// TIA Portal V18 export
FUNCTION "AHURegsAndTargetStatesInEconomyOpMode" : Void   // FC60031, LAD
{ S7_Optimized_Access := 'TRUE' }
VERSION : 0.1
// Operation Modes                                                 Unit State
// 0                                                                              0=Stopped
// 1=Economy                                                           1=Checking-up  
//                                                                                 2=Preheating
//                                                                                 3=Starting 
//                                                                                 4=RecirculatingOperation (Protection)
//                                                                                 5=Sustained Mode (Economy)
//                                                                                 Not 6=Sustained Mode (PreComfort setpoints) 
//                                                                                 Not 7=Comfort  operation
//                                                                                 Not 8=Night Cooling
//                                                                                 9=Stopping
//                                                                                 10=Blocking
//                                                                                 11=FrostProtecting
// stored: AutoNumber false, IsIECCheckEnabled false, SetENOAutomatically false, UDAEnableTagReadback false
   VAR_INPUT
      iUnitID : Int;
      cActualOpMode : Byte;
      cHeatingRegCfg : Byte;
      cCoolingRegCfg : Byte;
      cIAQRegCfg : Byte;
      cBuildingdPRegCfg : Byte;
   END_VAR
   VAR_OUTPUT
      cTargetState : Byte;
      cHeatingRegState : Byte;
      cCoolingRegState : Byte;
      cIAQRegState : Byte;
      cBuildingdPRegState : Byte;
   END_VAR
   VAR_TEMP
      SHTargetState : Int;
      SCTargetState : Int;
      SIAQTargetState : Int;
      SdPTargetState : Int;
   END_VAR
BEGIN

REGION Network 1: Sustained Heating
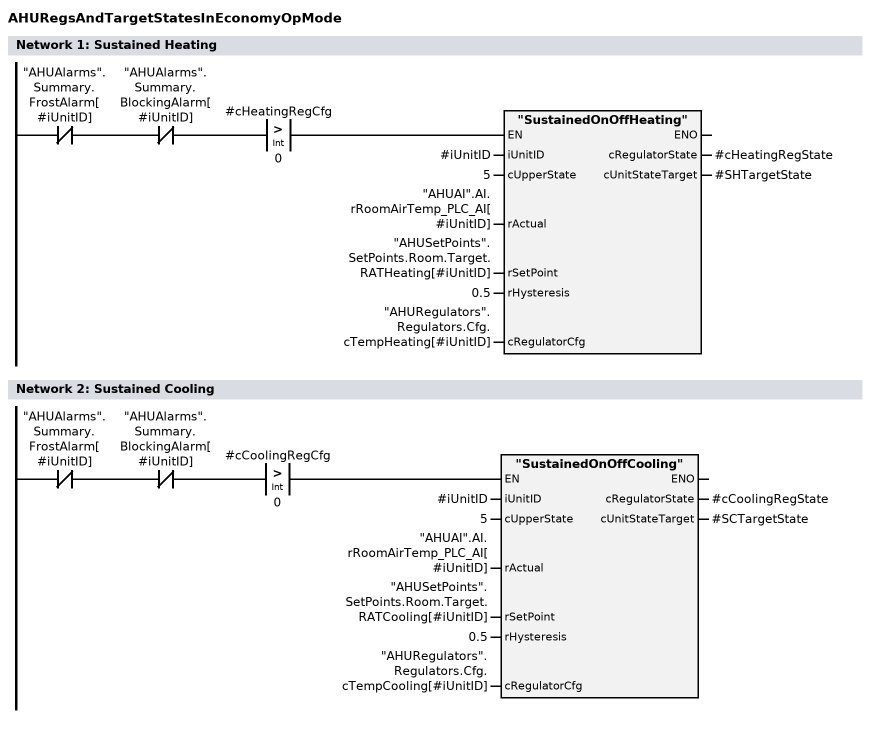
   RUNG wire#powerrail
      I_Contact( "AHUAlarms".Summary.FrostAlarm[#iUnitID] )
      I_Contact( "AHUAlarms".Summary.BlockingAlarm[#iUnitID] )
      { S7_Templates := "SrcType := Int" } GT_Contact(in1 := #cHeatingRegCfg, in2 := 0)
      "SustainedOnOffHeating"(iUnitID := #iUnitID, cUpperState := 5, rActual := "AHUAI".AI.rRoomAirTemp_PLC_AI[#iUnitID], rSetPoint := "AHUSetPoints".SetPoints.Room.Target.RATHeating[#iUnitID], rHysteresis := 0.5, cRegulatorCfg := "AHURegulators".Regulators.Cfg.cTempHeating[#iUnitID], cRegulatorState => #cHeatingRegState, cUnitStateTarget => #SHTargetState)
   END_RUNG
   // the same network as SCL:
   IF NOT "AHUAlarms".Summary.FrostAlarm[#iUnitID] AND NOT "AHUAlarms".Summary.BlockingAlarm[#iUnitID] AND (#cHeatingRegCfg > 0) THEN
       "SustainedOnOffHeating"(iUnitID := #iUnitID,
                               cUpperState := 5,
                               rActual := "AHUAI".AI.rRoomAirTemp_PLC_AI[#iUnitID],
                               rSetPoint := "AHUSetPoints".SetPoints.Room.Target.RATHeating[#iUnitID],
                               rHysteresis := 0.5,
                               cRegulatorCfg := "AHURegulators".Regulators.Cfg.cTempHeating[#iUnitID],
                               cRegulatorState => #cHeatingRegState,
                               cUnitStateTarget => #SHTargetState);
   END_IF;
END_REGION

REGION Network 2: Sustained Cooling
   RUNG wire#powerrail
      I_Contact( "AHUAlarms".Summary.FrostAlarm[#iUnitID] )
      I_Contact( "AHUAlarms".Summary.BlockingAlarm[#iUnitID] )
      { S7_Templates := "SrcType := Int" } GT_Contact(in1 := #cCoolingRegCfg, in2 := 0)
      "SustainedOnOffCooling"(iUnitID := #iUnitID, cUpperState := 5, rActual := "AHUAI".AI.rRoomAirTemp_PLC_AI[#iUnitID], rSetPoint := "AHUSetPoints".SetPoints.Room.Target.RATCooling[#iUnitID], rHysteresis := 0.5, cRegulatorCfg := "AHURegulators".Regulators.Cfg.cTempCooling[#iUnitID], cRegulatorState => #cCoolingRegState, cUnitStateTarget => #SCTargetState)
   END_RUNG
   // the same network as SCL:
   IF NOT "AHUAlarms".Summary.FrostAlarm[#iUnitID] AND NOT "AHUAlarms".Summary.BlockingAlarm[#iUnitID] AND (#cCoolingRegCfg > 0) THEN
       "SustainedOnOffCooling"(iUnitID := #iUnitID,
                               cUpperState := 5,
                               rActual := "AHUAI".AI.rRoomAirTemp_PLC_AI[#iUnitID],
                               rSetPoint := "AHUSetPoints".SetPoints.Room.Target.RATCooling[#iUnitID],
                               rHysteresis := 0.5,
                               cRegulatorCfg := "AHURegulators".Regulators.Cfg.cTempCooling[#iUnitID],
                               cRegulatorState => #cCoolingRegState,
                               cUnitStateTarget => #SCTargetState);
   END_IF;
END_REGION

REGION Network 3 (SCL)
   #cTargetState := INT_TO_BYTE(MAX(IN1 := #SHTargetState, IN2 := #SCTargetState));
END_REGION
END_FUNCTION
